// Mitsubishi GX Works2 project: PLC_GROUP24   PLC: FX3G

// global labels: Global1
VAR_GLOBAL
  Power_Off AT M1 : BOOL;
  Power_On AT X007 : BOOL;
  Work AT Y000 : BOOL;
  Mix_Start AT X003 : BOOL;
  Type_Word AT D1100 : REAL;
  Rand_Type AT D8280 : INT;
  Rand_TypeIN AT D7755 : INT;
  Continue1 AT M3 : BOOL;
END_VAR
VAR_GLOBAL CONSTANT
  Fivey : REAL := 5;
END_VAR
VAR_GLOBAL
  Protein_Snack AT M4 : BOOL;
  Classic_Snack AT M5 : BOOL;
  Input1 AT D1150 : REAL;
  Input2 AT D1160 : REAL;
  Input3 AT D1170 : REAL;
  Oats AT D2250 : REAL;
  Protain AT D2260 : REAL;
  Honey AT D2270 : REAL;
END_VAR
VAR_GLOBAL CONSTANT
  Con_Oats_P : REAL := 240;
  Con_Protain_P : REAL := 320;
END_VAR
VAR_GLOBAL
  Enough_Protein_Oats AT M6 : BOOL;
  Enough_Protein_protein AT M7 : BOOL;
END_VAR
VAR_GLOBAL CONSTANT
  Con_Honey_P : REAL := 160;
END_VAR
VAR_GLOBAL
  Enough_honey_Protein AT M8 : BOOL;
  Enough_PS AT M9 : BOOL;
END_VAR
VAR_GLOBAL CONSTANT
  Con_oats_C : REAL := 400;
END_VAR
VAR_GLOBAL
  Enough_Classic_Oats AT M10 : BOOL;
END_VAR
VAR_GLOBAL CONSTANT
  Con_Protain_C : REAL := 160;
END_VAR
VAR_GLOBAL
  Enough_Classic_Protein AT M11 : BOOL;
END_VAR
VAR_GLOBAL CONSTANT
  Con_Honey_C : REAL := 120;
END_VAR
VAR_GLOBAL
  Enough_CS AT M12 : BOOL;
END_VAR
VAR_GLOBAL CONSTANT
  Const_5 : INT := K50;
END_VAR
VAR_GLOBAL
  Mix_Timer AT TC9 : BOOL;
  Mix_Timer_ts9 AT TS9 : BOOL;
  Mix_Proccess AT Y003 : BOOL;
  Int_Snack AT D5000 : REAL;
END_VAR
VAR_GLOBAL CONSTANT
  Divide : REAL := 400;
END_VAR
VAR_GLOBAL
  SUB_P AT M14 : BOOL;
  S_Bakeing AT X002 : BOOL;
END_VAR
VAR_GLOBAL CONSTANT
  Time_For_CS : INT := 40;
END_VAR
VAR_GLOBAL
  Time_B AT D6000 : INT;
END_VAR
VAR_GLOBAL CONSTANT
  Time_For_PS : INT := 50;
END_VAR
VAR_GLOBAL
  Flash_Counter AT TC5 : BOOL;
  Flash_Counter_TC5 AT TS5 : BOOL;
  M_Y1 AT M36 : BOOL;
  Y1_Flash_Counter AT TC3 : BOOL;
END_VAR
VAR_GLOBAL CONSTANT
  Const_4 : INT := K4;
END_VAR
VAR_GLOBAL
  Timer_TS3 AT TS3 : BOOL;
  Y1_Light_On AT Y001 : BOOL;
  Y2_Flash_Counter AT TC4 : BOOL;
  Timer_TS4 AT TS4 : BOOL;
  Y2_Light_On AT Y002 : BOOL;
  SUB_C AT M15 : BOOL;
END_VAR
VAR_GLOBAL CONSTANT
  Const_10 : INT := K10;
END_VAR
VAR_GLOBAL
  Input_RES AT D1280 : REAL;
  C_mix AT M51 : BOOL;
  P_mix AT M41 : BOOL;
  Counter_Pack AT CC3 : BOOL;
  Pack_Start AT X006 : BOOL;
  Y4_Pack_Light AT Y004 : BOOL;
  CC3_T AT CS3 : BOOL;
  Unit_Pack AT X000 : BOOL;
END_VAR
VAR_GLOBAL CONSTANT
  Const_8 : INT := K8;
END_VAR
VAR_GLOBAL
  Pack_Counter AT D2025 : REAL;
END_VAR
VAR_GLOBAL CONSTANT
  P_Finish : REAL := 1.0;
END_VAR
VAR_GLOBAL
  EMO AT X005 : BOOL;
  End_Day_Light AT M50 : BOOL;
END_VAR
VAR_GLOBAL CONSTANT
  Const_40 : REAL := 40.0;
END_VAR
VAR_GLOBAL
  Pack_Mul AT D2035 : REAL;
  Analog_Output AT D8282 : INT;
  Start_Unit_Pack AT M37 : BOOL;
  Can_start AT M69 : BOOL;
  pause_mix AT M71 : BOOL;
  Can_start_oats AT M80 : BOOL;
  Can_start_honey AT M81 : BOOL;
  Can_start_protein AT M82 : BOOL;
  Help_Day_Light AT M3 : BOOL;
  Help_mix AT M3 : BOOL;
  Help_Day_L AT M85 : BOOL;
END_VAR

// task Task_01 (event TRUE, interval 0, priority 31): POU_01

PROGRAM POU_01
(* structured ladder/FBD written out as ST: instructions are called as NAME(EN, inputs, outputs); _pN, _eN, _tN stand for wires *)
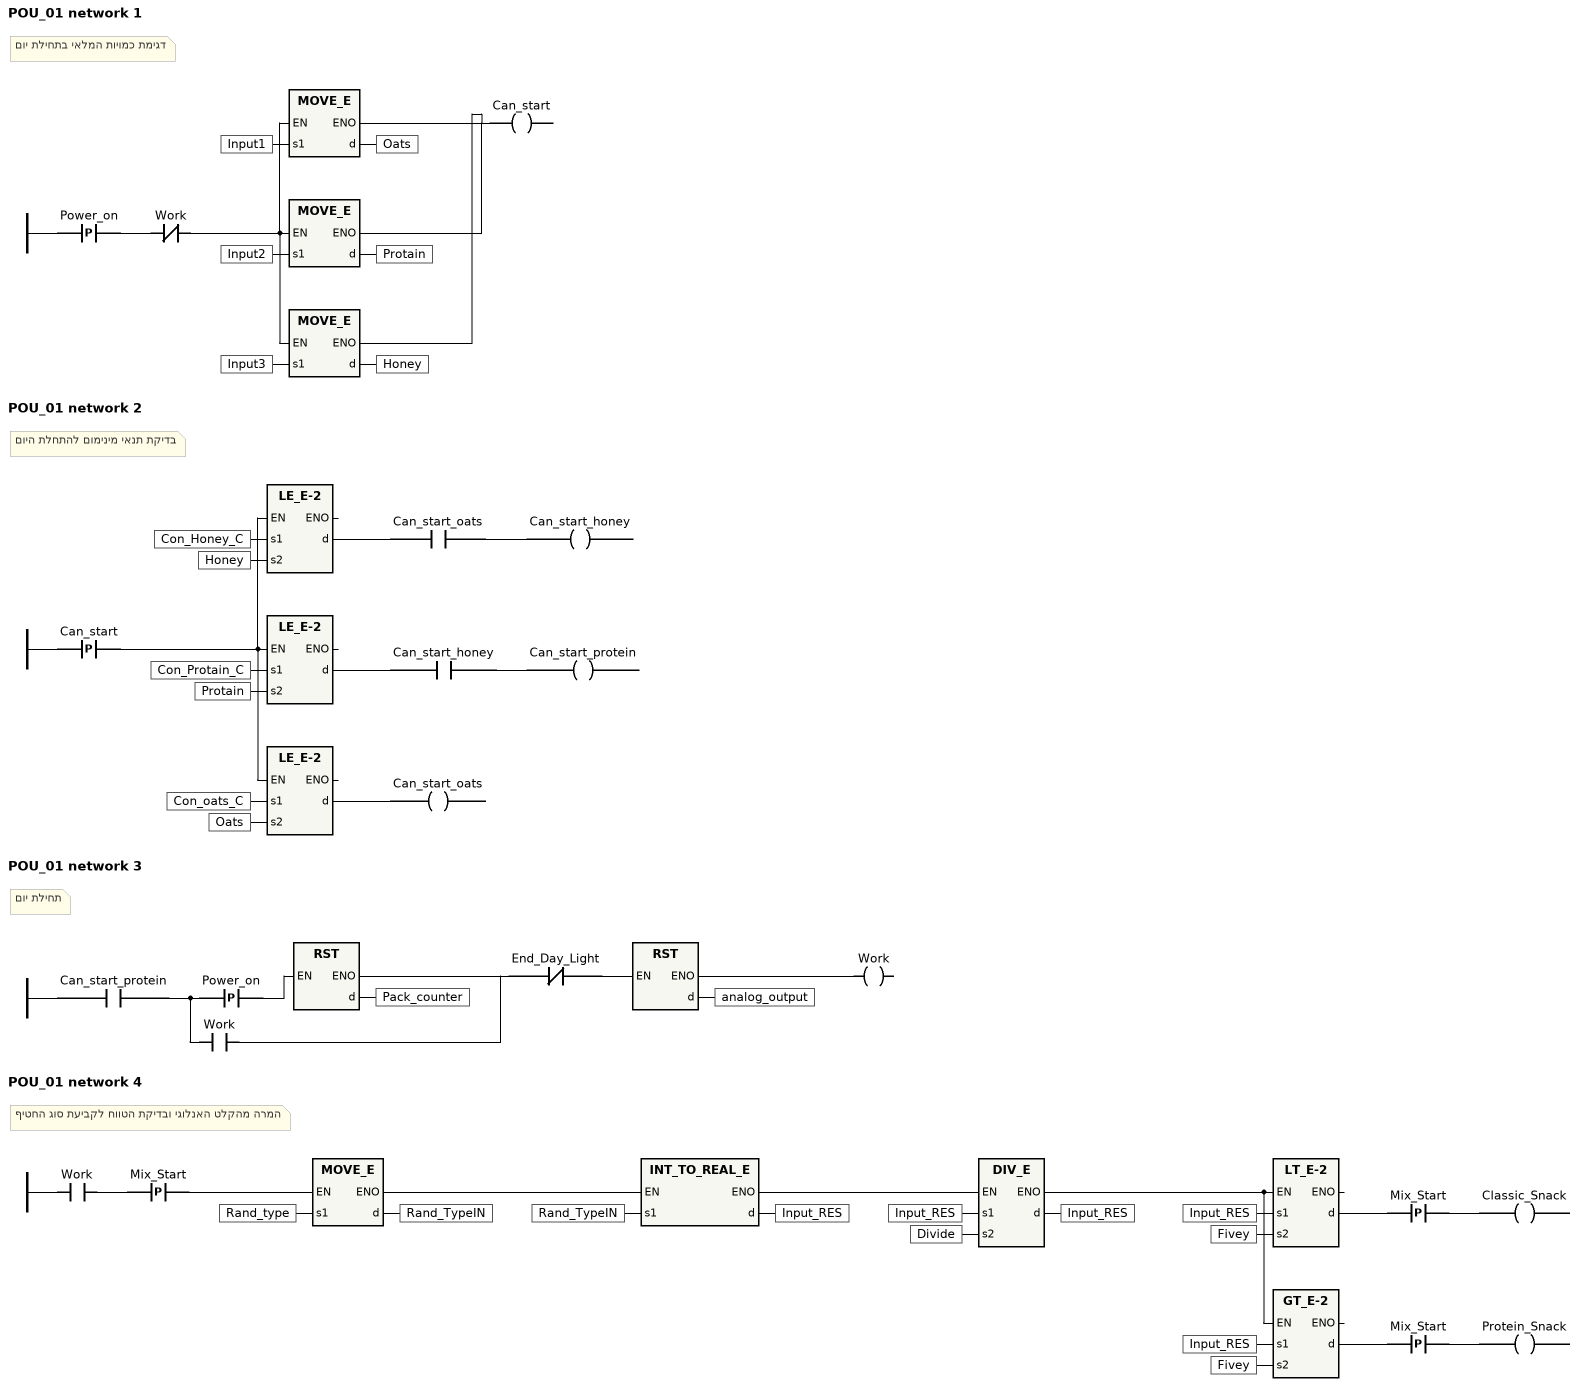
(* network 1 *)
(* דגימת כמויות המלאי בתחילת יום *)
_p1 := LDP(TRUE, Power_on) AND NOT Work;
_e2 := MOVE_E(_p1, Input1, Oats);
_e3 := MOVE_E(_p1, Input2, Protain);
_e4 := MOVE_E(_p1, Input3, Honey);
Can_start := _e2 OR _e3 OR _e4;
(* network 2 *)
(* בדיקת תנאי מינימום להתחלת היום *)
_p1 := LDP(TRUE, Can_start);
LE_E(_p1, Con_oats_C, Oats, _t2);
Can_start_oats := _t2;
LE_E(_p1, Con_Honey_C, Honey, _t3);
Can_start_honey := _t3 AND Can_start_oats;
LE_E(_p1, Con_Protain_C, Protain, _t4);
Can_start_protein := _t4 AND Can_start_honey;
(* network 3 *)
(* תחילת יום *)
_e1 := RST(Can_start_protein AND LDP(TRUE, Power_on), Pack_counter);
_e2 := RST((_e1 OR (Can_start_protein AND Work)) AND NOT End_Day_Light, analog_output);
Work := _e2;
(* network 4 *)
(* המרה מהקלט האנלוגי ובדיקת הטווח לקביעת סוג החטיף *)
_e1 := MOVE_E(Work AND LDP(TRUE, Mix_Start), Rand_type, Rand_TypeIN);
_e2 := INT_TO_REAL_E(_e1, Rand_TypeIN, Input_RES);
_e3 := DIV_E(_e2, Input_RES, Divide, Input_RES);
LT_E(_e3, Input_RES, Fivey, _t4);
Classic_Snack := _t4 AND LDP(TRUE, Mix_Start);
GT_E(_e3, Input_RES, Fivey, _t5);
Protein_Snack := _t5 AND LDP(TRUE, Mix_Start);
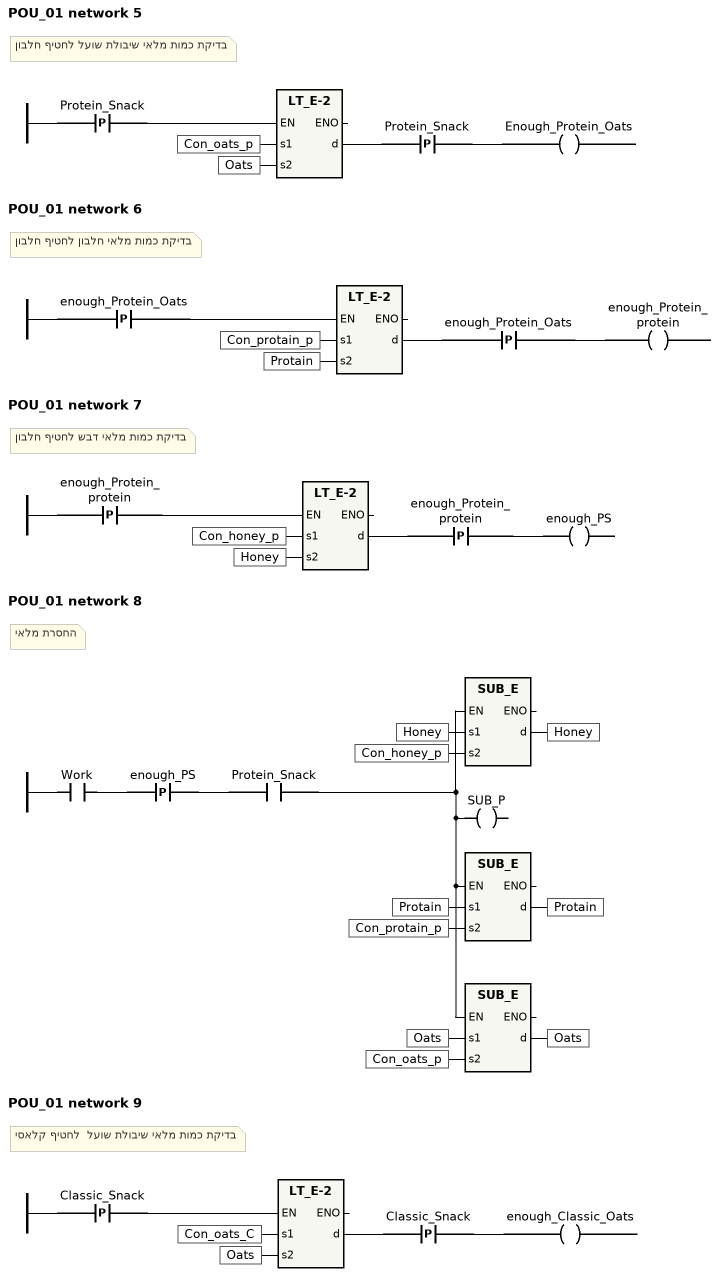
(* network 5 *)
(* בדיקת כמות מלאי שיבולת שועל לחטיף חלבון *)
LT_E(LDP(TRUE, Protein_Snack), Con_oats_p, Oats, _t1);
Enough_Protein_Oats := _t1 AND LDP(TRUE, Protein_Snack);
(* network 6 *)
(* בדיקת כמות מלאי חלבון לחטיף חלבון *)
LT_E(LDP(TRUE, enough_Protein_Oats), Con_protain_p, Protain, _t1);
enough_Protein_protein := _t1 AND LDP(TRUE, enough_Protein_Oats);
(* network 7 *)
(* בדיקת כמות מלאי דבש לחטיף חלבון *)
LT_E(LDP(TRUE, enough_Protein_protein), Con_honey_p, Honey, _t1);
enough_PS := _t1 AND LDP(TRUE, enough_Protein_protein);
(* network 8 *)
(* החסרת מלאי *)
_p1 := Work AND LDP(TRUE, enough_PS) AND Protein_Snack;
SUB_P := _p1;
SUB_E(_p1, Honey, Con_honey_p, Honey);
SUB_E(_p1, Protain, Con_protain_p, Protain);
SUB_E(_p1, Oats, Con_oats_p, Oats);
(* network 9 *)
(* בדיקת כמות מלאי שיבולת שועל  לחטיף קלאסי *)
LT_E(LDP(TRUE, Classic_Snack), Con_oats_C, Oats, _t1);
enough_Classic_Oats := _t1 AND LDP(TRUE, Classic_Snack);
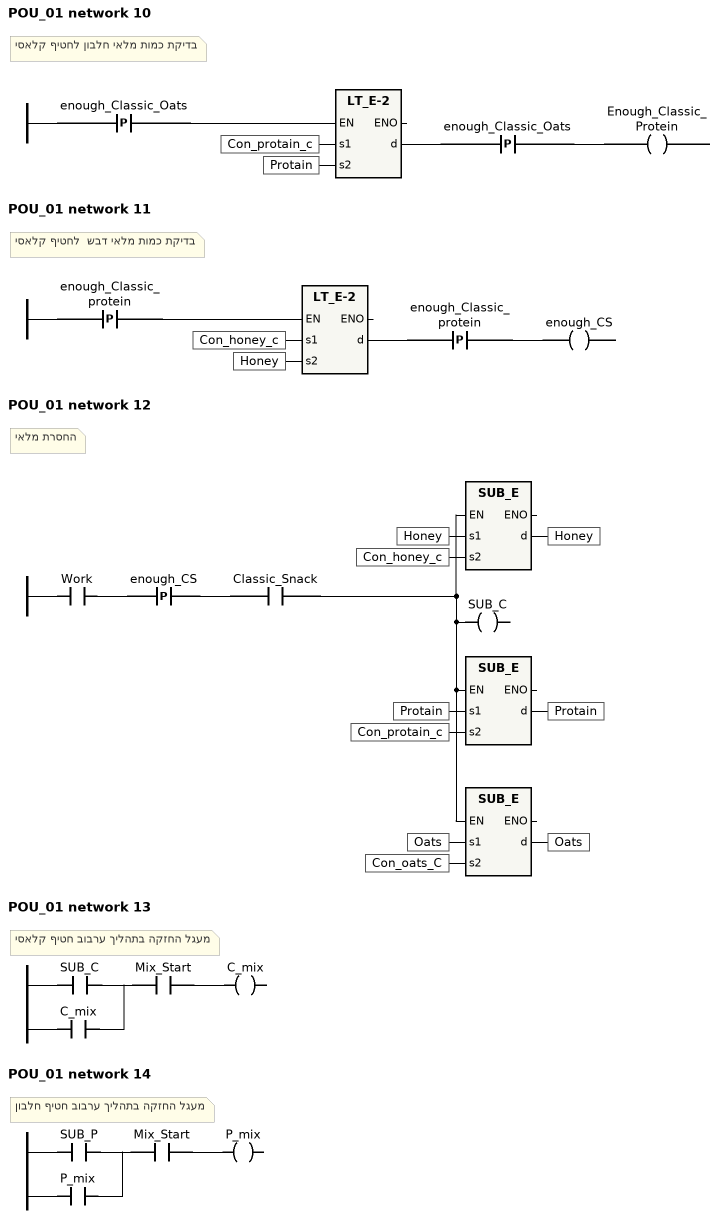
(* network 10 *)
(* בדיקת כמות מלאי חלבון לחטיף קלאסי *)
LT_E(LDP(TRUE, enough_Classic_Oats), Con_protain_c, Protain, _t1);
Enough_Classic_Protein := _t1 AND LDP(TRUE, enough_Classic_Oats);
(* network 11 *)
(* בדיקת כמות מלאי דבש  לחטיף קלאסי *)
LT_E(LDP(TRUE, enough_Classic_protein), Con_honey_c, Honey, _t1);
enough_CS := _t1 AND LDP(TRUE, enough_Classic_protein);
(* network 12 *)
(* החסרת מלאי *)
_p1 := Work AND LDP(TRUE, enough_CS) AND Classic_Snack;
SUB_C := _p1;
SUB_E(_p1, Honey, Con_honey_c, Honey);
SUB_E(_p1, Protain, Con_protain_c, Protain);
SUB_E(_p1, Oats, Con_oats_C, Oats);
(* network 13 *)
(* מעגל החזקה בתהליך ערבוב חטיף קלאסי *)
C_mix := (SUB_C OR C_mix) AND Mix_Start;
(* network 14 *)
(* מעגל החזקה בתהליך ערבוב חטיף חלבון *)
P_mix := (SUB_P OR P_mix) AND Mix_Start;
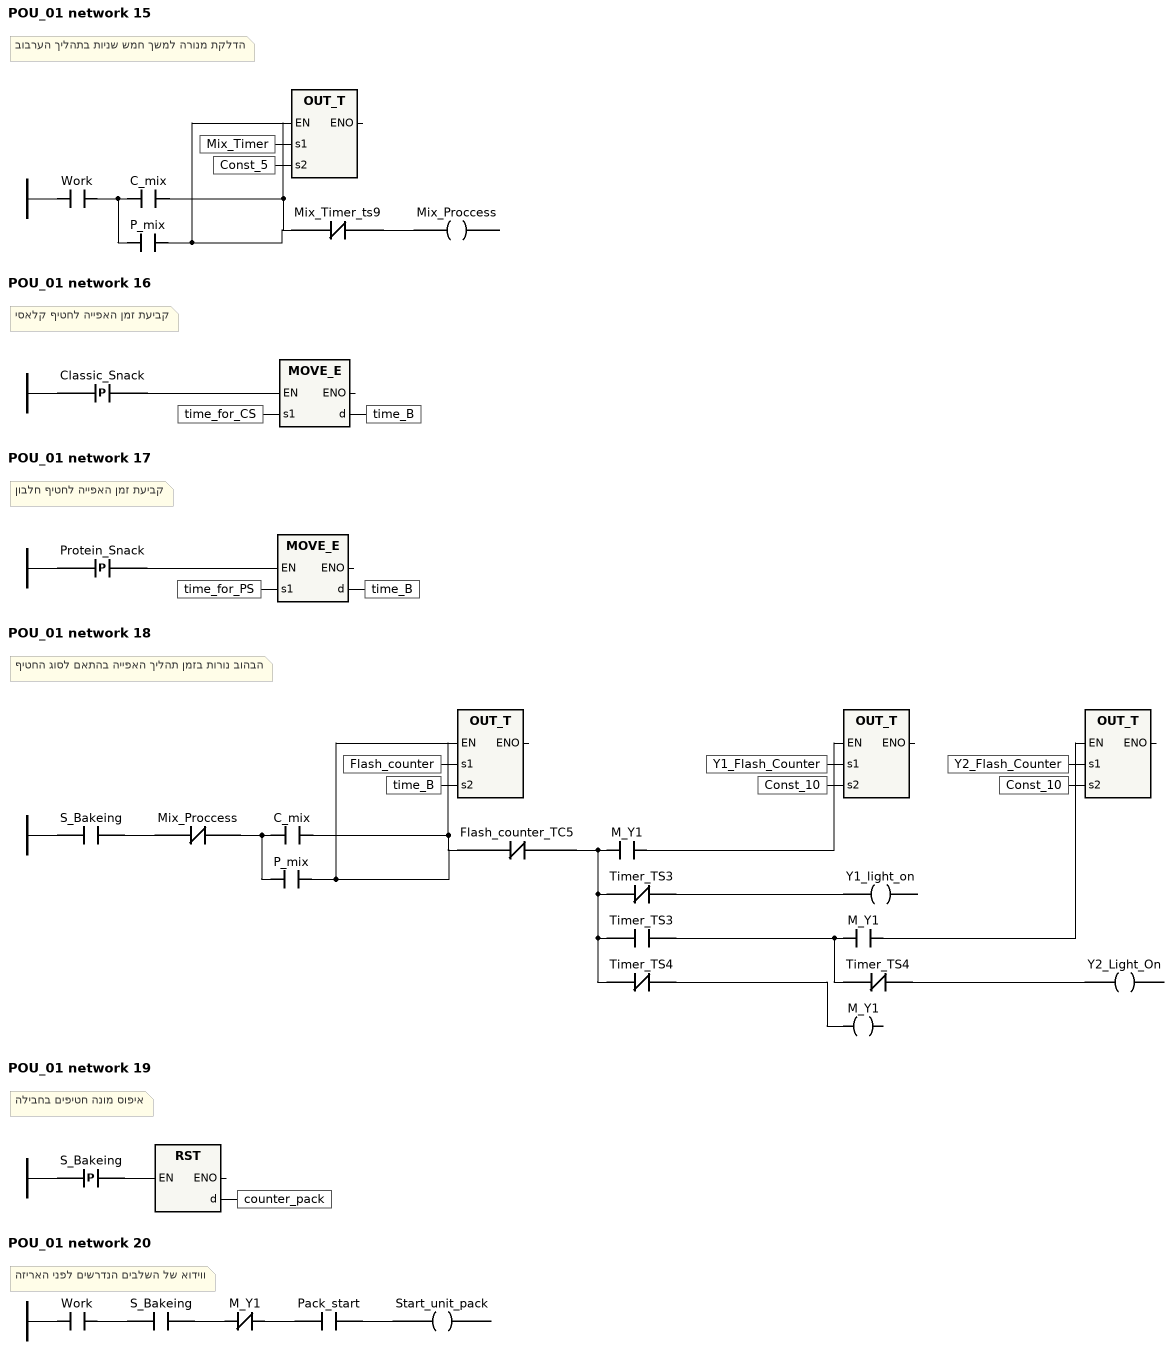
(* network 15 *)
(* הדלקת מנורה למשך חמש שניות בתהליך הערבוב *)
_p1 := (Work AND C_mix) OR (Work AND P_mix);
OUT_T(_p1, Mix_Timer, Const_5);
Mix_Proccess := _p1 AND NOT Mix_Timer_ts9;
(* network 16 *)
(* קביעת זמן האפייה לחטיף קלאסי *)
MOVE_E(LDP(TRUE, Classic_Snack), time_for_CS, time_B);
(* network 17 *)
(* קביעת זמן האפייה לחטיף חלבון *)
MOVE_E(LDP(TRUE, Protein_Snack), time_for_PS, time_B);
(* network 18 *)
(* הבהוב נורות בזמן תהליך האפייה בהתאם לסוג החטיף *)
_p1 := S_Bakeing AND NOT Mix_Proccess;
_p2 := (_p1 AND C_mix) OR (_p1 AND P_mix);
OUT_T(_p2, Flash_counter, time_B);
_p3 := _p2 AND NOT Flash_counter_TC5;
OUT_T(_p3 AND M_Y1, Y1_Flash_Counter, Const_10);
Y1_light_on := _p3 AND NOT Timer_TS3;
_p4 := _p3 AND Timer_TS3;
OUT_T(_p4 AND M_Y1, Y2_Flash_Counter, Const_10);
Y2_Light_On := _p4 AND NOT Timer_TS4;
M_Y1 := _p3 AND NOT Timer_TS4;
(* network 19 *)
(* איפוס מונה חטיפים בחבילה *)
RST(LDP(TRUE, S_Bakeing), counter_pack);
(* network 20 *)
(* ווידוא של השלבים הנדרשים לפני האריזה *)
Start_unit_pack := Work AND S_Bakeing AND NOT M_Y1 AND Pack_start;
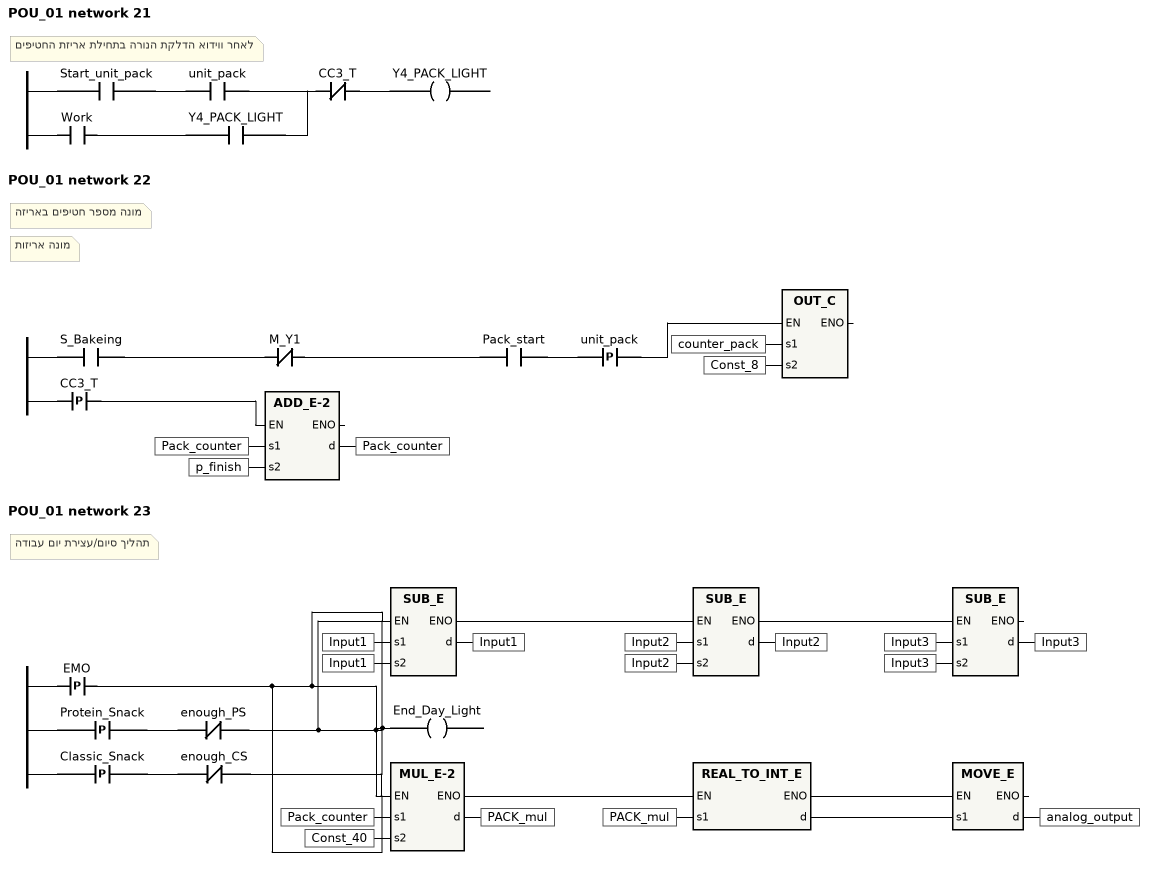
(* network 21 *)
(* לאחר ווידוא הדלקת הנורה בתחילת אריזת החטיפים *)
Y4_PACK_LIGHT := ((Start_unit_pack AND unit_pack) OR (Work AND Y4_PACK_LIGHT)) AND NOT CC3_T;
(* network 22 *)
(* מונה מספר חטיפים באריזה *)
(* מונה אריזות *)
OUT_C(S_Bakeing AND NOT M_Y1 AND Pack_start AND LDP(TRUE, unit_pack), counter_pack, Const_8);
ADD_E(LDP(TRUE, CC3_T), Pack_counter, p_finish, Pack_counter);
(* network 23 *)
(* תהליך סיום/עצירת יום עבודה *)
_p1 := LDP(TRUE, EMO) OR (LDP(TRUE, Protein_Snack) AND NOT enough_PS) OR (LDP(TRUE, Classic_Snack) AND NOT enough_CS);
End_Day_Light := _p1;
_e2 := SUB_E(_p1, Input1, Input1, Input1);
_e3 := SUB_E(_e2, Input2, Input2, Input2);
SUB_E(_e3, Input3, Input3, Input3);
_e4 := MUL_E(_p1, Pack_counter, Const_40, PACK_mul);
_e6 := REAL_TO_INT_E(_e4, PACK_mul, _t5);
MOVE_E(_e6, _t5, analog_output);
END_PROGRAM
